Staubli VAL3: SHR.pgx

public program SHR(num x_shift, num& x_value[])
// shift num value to left
begin
  if bDebug
    putln("SHR()")
  endIf
  x_value=roundDown(roundDown(x_value)/exp(roundDown(x_shift)*ln(2)))
end
